FUNCTION_BLOCK PermissiveInterlock IMPLEMENTS I_Permissive
VAR
	_OK				 : BOOL				   := TRUE;
	Permissive		 : ARRAY[0..9] OF BOOL := [TRUE, TRUE, TRUE, TRUE, TRUE, TRUE, TRUE, TRUE, TRUE, TRUE];
	PermissiveReason : ARRAY[0..9] OF STRING;
END_VAR

METHOD PROTECTED Check : BOOL
VAR
	i : UDINT;
END_VAR
_OK := TRUE;
FOR i := 0 TO 9 DO
	IF NOT Permissive[i] THEN
		_OK := FALSE;
	END_IF
END_FOR
END_METHOD

{attribute 'monitoring' := 'call'}
PROPERTY OK : BOOL
GET
OK := _OK;
END_GET
END_PROPERTY

METHOD Set
VAR_INPUT
	Index  : UDINT(0..9);
	Reason : STRING;
	Value  : BOOL;
END_VAR
Permissive[Index]		:= Value;
PermissiveReason[Index] := Reason;
Check();
END_METHOD

END_FUNCTION_BLOCK

(* stored: Version 1.1.0.1, ProductVersion 3.1.4026.18
   POU PermissiveInterlock: Id {3331978e-2c7e-4f0c-a7ff-432b8a75e3a8}, SpecialFunc None
   Method Check: Id {560987c4-f537-4ed7-ba95-bf7164c34026}
   Property OK: Id {b0b6552a-3a71-4f94-8697-8d20014ae9f0}
   Get Get: Id {4aea581a-fafb-4338-aea1-31b2ae2fd29e}
   Method Set: Id {ed65028d-a4f6-4770-b45a-73143a209f97} *)
